(* PLC project Tc2_Utilities.FB_GetDongleSystemID Demo, tc3-libraries-kb TwinCAT 3.1 *)
(* stored: creationDateTime 2026-05-10T20:00:00, modificationDateTime 2026-05-10T20:00:00 *)

PROGRAM P_Demo_FB_GetDongleSystemID
  VAR
    fbFB_GetDongleSystemID : FB_GetDongleSystemID;  (* Tc2_Utilities.FB_GetDongleSystemID 实例 *)
    arg_bExecute : BOOL;  (* VAR_INPUT bExecute *)
    arg_tTimeout : TIME;  (* VAR_INPUT tTimeout *)
    arg_sNetId : T_AmsNetId;  (* VAR_INPUT sNetId *)
    arg_stAmsAddr : AMSADDR;  (* VAR_INPUT stAmsAddr *)
    out_bBusy : BOOL;  (* VAR_OUTPUT bBusy *)
    out_bError : BOOL;  (* VAR_OUTPUT bError *)
    out_nErrorId : UDINT;  (* VAR_OUTPUT nErrorId *)
    out_stSystemID : GUID;  (* VAR_OUTPUT stSystemID *)
    out_stVolumeID : GUID;  (* VAR_OUTPUT stVolumeID *)
  END_VAR

            // ============================================================
// Tc2_Utilities.FB_GetDongleSystemID 演示程序（FB 实例）
// ============================================================
// 验证步骤：
//   1. 引用 Tc2_Utilities（及依赖类型所在库 Tc2_System 等）
//   2. 编译 + 登录
//   3. 按 doc.md 给 arg_* 赋值
//   4. 在线监视 out_* / io_* 输出
// ============================================================

fbFB_GetDongleSystemID(
    bExecute := arg_bExecute,
    tTimeout := arg_tTimeout,
    sNetId := arg_sNetId,
    stAmsAddr := arg_stAmsAddr,
    bBusy => out_bBusy,
    bError => out_bError,
    nErrorId => out_nErrorId,
    stSystemID => out_stSystemID,
    stVolumeID => out_stVolumeID
);

          
END_PROGRAM
